// TIA Portal V20 export
VAR_GLOBAL   // PLC tag table "Unit1Em5"
   "BA030AZSBK07.05" AT %I1024.5 : Bool;   // CATHODE MAIN P&P1 DETECT SENSOR
   "BA030AZSBK07.06" AT %I1024.6 : Bool;   // CATHODE MAIN P&P1 ROTARY CCW
   "BA030AZSBK07.07" AT %I1024.7 : Bool;   // CATHODE MAIN P&P1 PRESSURE SWITCH
   "BA030AZSBK07.16" AT %I1025.6 : Bool;   // CATHODE MAIN P&P1 ROTARY CW
   "BA030AZSBK08.03" AT %I1028.3 : Bool;   // CATHODE MAIN P&P2 DETECT SENSOR
   "BA030AZSBK08.04" AT %I1028.4 : Bool;   // CATHODE MAIN P&P2 PRESSURE SWITCH
   "BA030AZSBK13.06" AT %I1048.6 : Bool;   // CATHODE ALIGN TABLE ELECTRODE DETECT SENSOR
   "BA030AZSBK13.07" AT %I1048.7 : Bool;   // CATHODE ALIGN TABLE PRESSURE SWITCH
   "BA030AZSBK14.00" AT %I1052.0 : Bool;   // CATHODE FIX FRONT BACKWARD
   "BA030AZSBK14.02" AT %I1052.2 : Bool;   // CATHODE FIX REAR BACKWARD
   "BA030AZSBK14.04" AT %I1052.4 : Bool;   // FIX CATHODE DETECT SENSOR
   "BA030AZSBK14.10" AT %I1053.0 : Bool;   // CATHODE FIX FRONT FORWARD
   "BA030AZSBK14.12" AT %I1053.2 : Bool;   // CATHODE FIX REAR FORWARD
   "BA030AZSBK15.00" AT %I1056.0 : Bool;   // CATHODE NG BOX FULL SENSOR
   "BA030AZSBK15.01" AT %I1056.1 : Bool;   // CATHODE NG BOX NG BOX DETECT SENSOR
   "BA030AZSBK15.02" AT %I1056.2 : Bool;   // CATHODE NG BOX LIFT DOWN
   "BA030AZSBK15.03" AT %I1056.3 : Bool;   // CATHODE NG BOX LIFT UP
   "BA030AZSBK15.04" AT %I1056.4 : Bool;   // CATHODE NG BOX LOCK DOWN
   "BA030AZSBK15.05" AT %I1056.5 : Bool;   // CATHODE NG BOX LOCK UP
   "BA030AZSBK16.00" AT %I1060.0 : Bool;   // CATHODE MAIN NG P&P 1st BACKWARD
   "BA030AZSBK16.02" AT %I1060.2 : Bool;   // CATHODE MAIN NG P&P 2nd BACKWARD
   "BA030AZSBK16.04" AT %I1060.4 : Bool;   // CATHODE MAIN NG P&P UP
   "BA030AZSBK16.06" AT %I1060.6 : Bool;   // CATHODE NG P&P VACUUM PRESSURE SWITCH
   "BA030AZSBK16.10" AT %I1061.0 : Bool;   // CATHODE MAIN NG P&P 1st FORWARD
   "BA030AZSBK16.12" AT %I1061.2 : Bool;   // CATHODE MAIN NG P&P 2nd FORWARD
   "BA030AZSBK16.14" AT %I1061.4 : Bool;   // CATHODE MAIN NG P&P DOWN
   "BA030AZSBK16.16" AT %I1061.6 : Bool;   // CATHODE NG P&P ELECTRODE DETECT SENSOR
   "BA030AZSSP508.04" AT %I3002.4 : Bool;   // CATHODE ALIGN VISION BUSY (STO)
   "BA030AZSSP508.05" AT %I3002.5 : Bool;   // CATHODE ALIGN VISION READY (OK)
   "BA030AZSPM06.00" AT %Q2020.0 : Bool;   // CATHODE GLASS CLEANING ON
   "BA030AZSPM06.02" AT %Q2020.2 : Bool;   // CATHODE MAIN NG P&P DOWN
   "BA030AZSPM06.03" AT %Q2020.3 : Bool;   // CATHODE MAIN NG P&P UP
   "BA030AZSPM06.04" AT %Q2020.4 : Bool;   // CATHODE MAIN NG P&P 1st FORWARD
   "BA030AZSPM06.05" AT %Q2020.5 : Bool;   // CATHODE MAIN NG P&P 1st BACKWARD
   "BA030AZSPM06.06" AT %Q2020.6 : Bool;   // CATHODE MAIN NG P&P 2nd FORWARD
   "BA030AZSPM06.07" AT %Q2020.7 : Bool;   // CATHODE MAIN NG P&P 2nd BACKWARD
   "BA030AZSPM06.10" AT %Q2021.0 : Bool;   // CATHODE FIX FRONT&REAR FORWARD
   "BA030AZSPM06.11" AT %Q2021.1 : Bool;   // CATHODE FIX FRONT&REAR BACKWARD
   "BA030AZSPM06.12" AT %Q2021.2 : Bool;   // CATHODE MAIN P&P#1 ROTARY CW
   "BA030AZSPM06.13" AT %Q2021.3 : Bool;   // CATHODE MAIN P&P#1 ROTARY CCW
   "BA030AZSPM06.14" AT %Q2021.4 : Bool;   // CATHODE NG BOX LIFT UP
   "BA030AZSPM06.15" AT %Q2021.5 : Bool;   // CATHODE NG BOX LIFT DOWN
   "BA030AZSPM06.16" AT %Q2021.6 : Bool;   // CATHODE NG BOX LOCK UP
   "BA030AZSPM06.17" AT %Q2021.7 : Bool;   // CATHODE NG BOX LOCK DOWN
   "BA030AZSBK32.00" AT %Q2204.0 : Bool;   // CATHODE MAIN P&P1 VACUUM ON
   "BA030AZSBK32.01" AT %Q2204.1 : Bool;   // CATHODE MAIN P&P1 VACUUM OFF
   "BA030AZSBK32.02" AT %Q2204.2 : Bool;   // CATHODE MAIN P&P2 VACUUM ON
   "BA030AZSBK32.03" AT %Q2204.3 : Bool;   // CATHODE MAIN P&P2 VACUUM OFF
   "BA030AZSBK32.04" AT %Q2204.4 : Bool;   // CATHODE MAIN NG P&P VACUUM ON
   "BA030AZSBK32.05" AT %Q2204.5 : Bool;   // CATHODE MAIN NG P&P VACUUM OFF
   "BA030AZSBK32.06" AT %Q2204.6 : Bool;   // CATHODE ALIGN TABLE VACUUM ON
   "BA030AZSBK32.07" AT %Q2204.7 : Bool;   // CATHODE ALIGN TABLE VACUUM OFF
   "BA030AZSPM01.16" AT %Q2001.6 : Bool;   // CATHODE CONVEYOR PICK UP ON
   "BA030AZSPM07.16" AT %Q2025.6 : Bool;   // CATHODE CONVEYOR COVER FORWARD
   "BA030AZSPM07.17" AT %Q2025.7 : Bool;   // CATHODE CONVEYOR COVER BACKWARD
   "BA030AZSSP504.14" AT %Q3300.4 : Bool;   // CATHODE ALIGN VISION CONTROLLER TRIGEER IN
END_VAR
VAR_GLOBAL CONSTANT   // user constants
   U1EM5_JOB01 : DInt := 1;
   U1EM5_JOB02 : DInt := 2;
   U1EM5_JOB03 : DInt := 3;
   U1EM5_JOB04 : DInt := 4;
   U1EM5_JOB05 : DInt := 5;
   U1EM5_JOB06 : DInt := 6;
   U1EM5_JOB07 : DInt := 7;
   U1EM5_JOB08 : DInt := 8;
   U1EM5_JOB09 : DInt := 9;
   U1EM5_JOB10 : DInt := 10;
   U1EM5_JOB11 : DInt := 11;
   U1EM5_JOB12 : DInt := 12;
   U1EM5_JOB13 : DInt := 13;
   U1EM5_JOB14 : DInt := 14;
   U1EM5_JOB15 : DInt := 15;
   U1EM5_JOB16 : DInt := 16;
   U1EM5_JOB17 : DInt := 17;
   U1EM5_JOB18 : DInt := 18;
   U1EM5_JOB19 : DInt := 19;
   U1EM5_JOB20 : DInt := 20;
   U1EM5_JOB21 : DInt := 21;
   U1EM5_JOB22 : DInt := 22;
   U1EM5_JOB23 : DInt := 23;
   U1EM5_JOB24 : DInt := 24;
   U1EM5_JOB25 : DInt := 25;
   U1EM5_JOB26 : DInt := 26;
   U1EM5_JOB27 : DInt := 27;
   U1EM5_JOB28 : DInt := 28;
   U1EM5_JOB29 : DInt := 29;
   U1EM5_JOB30 : DInt := 30;
   U1EM5_JOB31 : DInt := 31;
   U1EM5_JOB32 : DInt := 32;
   U1EM5_JOB33 : DInt := 33;
   U1EM5_JOB34 : DInt := 34;
   U1EM5_JOB35 : DInt := 35;
   U1EM5_JOB36 : DInt := 36;
   U1EM5_JOB37 : DInt := 37;
   U1EM5_JOB38 : DInt := 38;
   U1EM5_JOB39 : DInt := 39;
   U1EM5_JOB40 : DInt := 40;
   U1EM5_JOB41 : DInt := 41;
   U1EM5_JOB42 : DInt := 42;
   U1EM5_JOB43 : DInt := 43;
   U1EM5_JOB44 : DInt := 44;
   U1EM5_JOB45 : DInt := 45;
   U1EM5_JOB46 : DInt := 46;
   U1EM5_JOB47 : DInt := 47;
   U1EM5_JOB48 : DInt := 48;
   U1EM5_JOB49 : DInt := 49;
   U1EM5_JOB50 : DInt := 50;
   U1EM5_JOB51 : DInt := 51;
   U1EM5_JOB52 : DInt := 52;
   U1EM5_JOB53 : DInt := 53;
   U1EM5_JOB54 : DInt := 54;
   U1EM5_JOB55 : DInt := 55;
   U1EM5_JOB56 : DInt := 56;
   U1EM5_JOB57 : DInt := 57;
   U1EM5_JOB58 : DInt := 58;
   U1EM5_JOB59 : DInt := 59;
   U1EM5_JOB60 : DInt := 60;
   U1EM5_JOB61 : DInt := 61;
   U1EM5_JOB62 : DInt := 62;
   U1EM5_JOB63 : DInt := 63;
   U1EM5_JOB64 : DInt := 64;
   U1EM5_JOB65 : DInt := 65;
   U1EM5_JOB66 : DInt := 66;
   U1EM5_JOB67 : DInt := 67;
   U1EM5_JOB68 : DInt := 68;
   U1EM5_JOB69 : DInt := 69;
   U1EM5_JOB70 : DInt := 70;
   U1EM5_JOB71 : DInt := 71;
   U1EM5_JOB72 : DInt := 72;
   U1EM5_JOB73 : DInt := 73;
   U1EM5_JOB74 : DInt := 74;
   U1EM5_JOB75 : DInt := 75;
   U1EM5_JOB76 : DInt := 76;
   U1EM5_JOB77 : DInt := 77;
   U1EM5_JOB78 : DInt := 78;
   U1EM5_JOB79 : DInt := 79;
   U1EM5_JOB80 : DInt := 80;
   U1EM5_JOB81 : DInt := 81;
   U1EM5_JOB82 : DInt := 82;
   U1EM5_JOB83 : DInt := 83;
   U1EM5_JOB84 : DInt := 84;
   U1EM5_JOB85 : DInt := 85;
   U1EM5_JOB86 : DInt := 86;
   U1EM5_JOB87 : DInt := 87;
   U1EM5_JOB88 : DInt := 88;
   U1EM5_JOB89 : DInt := 89;
   U1EM5_JOB90 : DInt := 90;
   U1EM5_JOB91 : DInt := 91;
   U1EM5_JOB92 : DInt := 92;
   U1EM5_JOB93 : DInt := 93;
   U1EM5_JOB94 : DInt := 94;
   U1EM5_JOB95 : DInt := 95;
   U1EM5_JOB96 : DInt := 96;
   U1EM5_JOB97 : DInt := 97;
   U1EM5_JOB98 : DInt := 98;
   U1EM5_JOB99 : DInt := 99;
   U1EM5_SEQUENCE01 : Int := 1;
   U1EM5_SEQUENCE02 : Int := 2;
   U1EM5_SEQUENCE03 : Int := 3;
   U1EM5_SEQUENCE04 : Int := 4;
   U1EM5_SEQUENCE05 : Int := 5;
   U1EM5_SEQUENCE06 : Int := 6;
   U1EM5_SEQUENCE07 : Int := 7;
   U1EM5_SEQUENCE08 : Int := 8;
   U1EM5_SEQUENCE09 : Int := 9;
   U1EM5_SEQUENCE10 : Int := 10;
   U1EM5_SEQUENCE11 : Int := 11;
   U1EM5_SEQUENCE12 : Int := 12;
   U1EM5_SEQUENCE13 : Int := 13;
   U1EM5_SEQUENCE14 : Int := 14;
   U1EM5_SEQUENCE15 : Int := 15;
   U1EM5_SEQUENCE16 : Int := 16;
   U1EM5_SEQUENCE17 : Int := 17;
   U1EM5_SEQUENCE18 : Int := 18;
   U1EM5_SEQUENCE19 : Int := 19;
   U1EM5_SEQUENCE20 : Int := 20;
   U1EM5_SEQUENCE21 : Int := 21;
   U1EM5_SEQUENCE22 : Int := 22;
   U1EM5_SEQUENCE23 : Int := 23;
   U1EM5_SEQUENCE24 : Int := 24;
   U1EM5_SEQUENCE25 : Int := 25;
   U1EM5_SEQUENCE26 : Int := 26;
   U1EM5_SEQUENCE27 : Int := 27;
   U1EM5_SEQUENCE28 : Int := 28;
   U1EM5_SEQUENCE29 : Int := 29;
   U1EM5_SEQUENCE30 : Int := 30;
   U1EM5_SEQUENCE31 : Int := 31;
   U1EM5_SEQUENCE32 : Int := 32;
   U1EM5_SEQUENCE33 : Int := 33;
   U1EM5_SEQUENCE34 : Int := 34;
   U1EM5_SEQUENCE35 : Int := 35;
   U1EM5_SEQUENCE36 : Int := 36;
   U1EM5_SEQUENCE37 : Int := 37;
   U1EM5_SEQUENCE38 : Int := 38;
   U1EM5_SEQUENCE39 : Int := 39;
   U1EM5_SEQUENCE40 : Int := 40;
   U1EM5_SEQUENCE41 : Int := 41;
   U1EM5_SEQUENCE42 : Int := 42;
   U1EM5_SEQUENCE43 : Int := 43;
   U1EM5_SEQUENCE44 : Int := 44;
   U1EM5_SEQUENCE45 : Int := 45;
   U1EM5_SEQUENCE46 : Int := 46;
   U1EM5_SEQUENCE47 : Int := 47;
   U1EM5_SEQUENCE48 : Int := 48;
   U1EM5_SEQUENCE49 : Int := 49;
   U1EM5_SEQUENCE50 : Int := 50;
   U1EM5_SEQUENCE51 : Int := 51;
   U1EM5_SEQUENCE52 : Int := 52;
   U1EM5_SEQUENCE53 : Int := 53;
   U1EM5_SEQUENCE54 : Int := 54;
   U1EM5_SEQUENCE55 : Int := 55;
   U1EM5_SEQUENCE56 : Int := 56;
   U1EM5_SEQUENCE57 : Int := 57;
   U1EM5_SEQUENCE58 : Int := 58;
   U1EM5_SEQUENCE59 : Int := 59;
   U1EM5_SEQUENCE60 : Int := 60;
   U1EM5_SEQUENCE61 : Int := 61;
   U1EM5_SEQUENCE62 : Int := 62;
   U1EM5_SEQUENCE63 : Int := 63;
   U1EM5_SEQUENCE64 : Int := 64;
   U1EM5_SEQUENCE65 : Int := 65;
   U1EM5_SEQUENCE66 : Int := 66;
   U1EM5_SEQUENCE67 : Int := 67;
   U1EM5_SEQUENCE68 : Int := 68;
   U1EM5_SEQUENCE69 : Int := 69;
   U1EM5_SEQUENCE70 : Int := 70;
   U1EM5_SEQUENCE71 : Int := 71;
   U1EM5_SEQUENCE72 : Int := 72;
   U1EM5_SEQUENCE73 : Int := 73;
   U1EM5_SEQUENCE74 : Int := 74;
   U1EM5_SEQUENCE75 : Int := 75;
   U1EM5_SEQUENCE76 : Int := 76;
   U1EM5_SEQUENCE77 : Int := 77;
   U1EM5_SEQUENCE78 : Int := 78;
   U1EM5_SEQUENCE79 : Int := 79;
   U1EM5_SEQUENCE80 : Int := 80;
   U1EM5_SEQUENCE81 : Int := 81;
   U1EM5_SEQUENCE82 : Int := 82;
   U1EM5_SEQUENCE83 : Int := 83;
   U1EM5_SEQUENCE84 : Int := 84;
   U1EM5_SEQUENCE85 : Int := 85;
   U1EM5_SEQUENCE86 : Int := 86;
   U1EM5_SEQUENCE87 : Int := 87;
   U1EM5_SEQUENCE88 : Int := 88;
   U1EM5_SEQUENCE89 : Int := 89;
   U1EM5_SEQUENCE90 : Int := 90;
   U1EM5_SEQUENCE91 : Int := 91;
   U1EM5_SEQUENCE92 : Int := 92;
   U1EM5_SEQUENCE93 : Int := 93;
   U1EM5_SEQUENCE94 : Int := 94;
   U1EM5_SEQUENCE95 : Int := 95;
   U1EM5_SEQUENCE96 : Int := 96;
   U1EM5_SEQUENCE97 : Int := 97;
   U1EM5_SEQUENCE98 : Int := 98;
   U1EM5_SEQUENCE99 : Int := 99;
   U1EM5_NO_OF_SEQUENCE : USInt := 3;
   U1EM5_NO_OF_AXES : USInt := 8;
   U1EM5_NO_OF_CAM : USInt := 4;
   U1EM5_NO_OF_OUTPUTCAM : USInt := 22;
END_VAR
